{attribute 'no_explicit_call' := 'Do not call this POU directly'}
FUNCTION_BLOCK FB_HE_SolidAttenuatorFilterConstantThickness EXTENDS FB_Fallible IMPLEMENTS I_HE_SolidAttenuatorFilter
VAR
    iConvertUnits : I_ConvertUnitsLREAL;
    iCenterPointInAxisCoordinates : I_QuantityLREAL;
    fbLength : FB_QuantityLREALPublic(Units := 'mm');
    fbThickness : FB_QuantityLREALPublic(Units := 'um');
    sMaterial : T_MaxString;

    fbQueryPointInAxisCoordinates : FB_QuantityLREALPublic(Units := 'mm');
END_VAR


METHOD FB_Init: BOOL
VAR_INPUT
    bInitRetains: BOOL; // TRUE: the retain variables are initialized (reset warm / reset cold)
    bInCopyCode: BOOL;  // TRUE: the instance will be copied to the copy code afterward (online change)

    ConvertUnits : I_ConvertUnitsLREAL;
    CenterPointInAxisCoordinates : I_QuantityLREAL;
    Length : LREAL; // [mm]
    Thickness : LREAL; // [um]
    Material : T_MaxString;
END_VAR

iConvertUnits := ConvertUnits;
iCenterPointInAxisCoordinates := CenterPointInAxisCoordinates;
fbLength.Val := Length;
fbThickness.Val := Thickness;
sMaterial := Material;
END_METHOD


METHOD GetCenterPosition
VAR_INPUT
    CenterPosition : I_QuantityLREALPublic;
END_VAR

CenterPosition.Copy(QuantityToCopy := iCenterPointInAxisCoordinates);
END_METHOD


METHOD GetLength
VAR_INPUT
    Length : I_QuantityLREALPublic;
END_VAR

Length.Copy(QuantityToCopy := fbLength);
END_METHOD


METHOD GetMaterial
VAR_IN_OUT
    Material : T_MaxString;
END_VAR

Material := sMaterial;
END_METHOD


METHOD GetThicknessAt
VAR_INPUT
    QueryPointInAxisCoordinates : I_QuantityLREAL;
    Thickness : I_QuantityLREALPublic;
END_VAR

iConvertUnits.ConvertQuantityLREAL(
    QuantityToConvert := QueryPointInAxisCoordinates,
    DesiredUnits := iCenterPointInAxisCoordinates.Units,
    ConvertedQuantity := fbQueryPointInAxisCoordinates
);

IF iConvertUnits.GetError() THEN
    SetError(Msg := 'Query point units are invalid.');
    Thickness.SetError(Msg := GetErrorMsg());
END_IF

IF ABS(fbQueryPointInAxisCoordinates.Val - iCenterPointInAxisCoordinates.Val) <= fbLength.Val / 2.0 THEN
    // Query point is on the filter
    Thickness.Copy(QuantityToCopy := fbThickness);
ELSE
    // Query point is not on the filter
    Thickness.Copy(QuantityToCopy := fbThickness);
    Thickness.Val := 0.0;
END_IF
END_METHOD

END_FUNCTION_BLOCK

(* stored: Version 1.1.0.1
   POU FB_HE_SolidAttenuatorFilterConstantThickness: Id {530a2b44-a718-418a-ac99-1c6da73f59f7}, SpecialFunc None
   Method FB_Init: Id {78df13ab-eeec-4a22-b20c-16d636b1efe1}
   Method GetCenterPosition: Id {e24f7fba-26d8-4d1c-9b53-e7bf5c2c6a6d}
   Method GetLength: Id {12fdf4c3-b0b3-43c7-bae0-0b8d4ea07dc2}
   Method GetMaterial: Id {51489bc2-13c4-48c0-a8d0-03ddb1b7fa70}
   Method GetThicknessAt: Id {b8f52c11-4c90-4350-b5ab-2bc520fdef51} *)
